// TIA Portal project "ISA_navidad" (V16)

(* hardware
DEVICE "S7-1200 station_1"  S7-1200 Station
   slot 0: "Rack_0"  S7-1200 Rack  Rack  V1.0
   slot 1: "PLC_1"  CPU 1215C DC/DC/DC  6ES7 215-1AG40-0XB0  V4.4
DEVICE "SINAMICS G_1"  Sinamics.Device
   slot 0: "	_0"  Rail  SinamicsG120RackPN
   slot 0: "Accionamiento_1"  G120 CU240E-2 PN  6SL3244-0BB12-1FA0  4.7.10
      slot 1: "Interfaz PROFINET"  MDD-SinamicsG120-P
   slot 3: "PM240 IP20"  PM240 IP20  6SL3224-0BE13-7UA0  -
DEVICE "PC-System_1"  SIMATIC PC station
   slot 0: "Estación PC SIMATIC"  Rail  SIMATIC PC-Station  V1.0
      slot 125: "Stationmanager"  Station_Manager  V6.0.4
   slot 1: "HMI_RT_1"  WinCC RT Advanced  6AV2 104-0xxxx-xxxx  16.0.0.0
      slot 33792: "Interfaz del equipo"  Host interface
   slot 2: "IE general_1"  IE General  IE_CP  V8.2.0
*)

// ===== PLC "PLC_1"  CPU 1215C DC/DC/DC =====

VAR_GLOBAL   // PLC tag table "Tabla de variables estándar"
   "marcha_pulsador" AT %I0.0 : Bool;   // S1
   "paro_pulsador" AT %I0.1 : Bool;   // S2
   "emergencia_pulsador" AT %I0.2 : Bool;   // S3
   "funcionamiento_variador" AT %I0.5 : Bool;   // DO1+ (Motor girando)
   "aviso_activo_variador" AT %I0.6 : Bool;   // DO2+ (Variador en fallo)
   "temperatura_sensor" AT %IW64 : Int;   // B4
   "nivel_sensor" AT %IW66 : Int;   // B5
   "marcha_variador" AT %Q0.0 : Bool;
   "verde_piloto" AT %Q0.1 : Bool;   // H1
   "rojo_piloto" AT %Q0.2 : Bool;   // H2
   "ambar_piloto" AT %Q0.3 : Bool;   // H3
   "electrovalvula_1" AT %Q0.6 : Bool;   // Y1
   "electrovalvula_2" AT %Q0.7 : Bool;   // Y2
   "electrovalvula_3" AT %Q1.0 : Bool;   // Y3
   "resistencia_calefactora" AT %QW64 : Int;   // R1
   "frecuencia_variador" AT %QW66 : Int;
   "etapa_0" AT %M10.0 : Bool;
   "etapa_1" AT %M10.1 : Bool;
   "etapa_2" AT %M10.2 : Bool;
   "etapa_3" AT %M10.3 : Bool;
   "etapa_4" AT %M10.4 : Bool;
   "etapa_5" AT %M10.5 : Bool;
   "etapa_10" AT %M11.0 : Bool;
   "etapa_11" AT %M11.1 : Bool;
   "etapa_12" AT %M11.2 : Bool;
   "principal_etapas" AT %MB10 : Byte;   // Etapas 0 a 5
   "System_Byte" AT %MB1 : Byte;
   "FirstScan" AT %M1.0 : Bool;
   "DiagStatusUpdate" AT %M1.1 : Bool;
   "AlwaysTRUE" AT %M1.2 : Bool;
   "AlwaysFALSE" AT %M1.3 : Bool;
   "Clock_Byte" AT %MB0 : Byte;
   "Clock_10Hz" AT %M0.0 : Bool;
   "Clock_5Hz" AT %M0.1 : Bool;
   "Clock_2.5Hz" AT %M0.2 : Bool;
   "Clock_2Hz" AT %M0.3 : Bool;
   "Clock_1.25Hz" AT %M0.4 : Bool;
   "Clock_1Hz" AT %M0.5 : Bool;
   "Clock_0.625Hz" AT %M0.6 : Bool;
   "Clock_0.5Hz" AT %M0.7 : Bool;
END_VAR

DATA_BLOCK "Variables"   // DB1
{ S7_Optimized_Access := 'TRUE' }
VERSION : 0.1
   VAR
      T1_PT : Time;   // PT de T1 convertido a segundos
      T2_PT : Time;   // PT de T2 convertido a segundos
      Setpoint_PID : Real;   // Setpoint del PID
      temperatura_escalada : Real;   // Temperatura escalada [0..100]ºC
      mode_PID : Int;   // Modo de funcionamiento PID
      mode_activate_PID : Bool;   // Activación del modo de PID
      output_PID : Real;   // Salida del PID [0..100]%
      nivel_escalado : Real;   // Nivel del tanque escalado [0..75] litros
      velocidad_lenta_SCADA : Int;   // Frecuencia lenta seleccionada en SCADA
      velocidad_rapida_SCADA : Int;   // Frecuencia rápida seleccionada en SCADA
      consigna_velocidad : Int;   // Consigna de frecuencia del variador
      paro_SCADA : Bool;   // Pulsador de paro en SCADA
      marcha_SCADA : Bool;   // Pulsador de marcha en SCADA
      estado_motor_scada : Bool;   // Piloto estado motor SCADA
      paro_emergencia_SCADA : Bool;   // Paro de emergencia SCADA
      piloto_velocidad_lenta_SCADA : Bool;   // Piloto de velocidad lenta SCADA
      piloto_velocidad_rapida_SCADA : Bool;   // Piloto de velocidad rápida SCADA
      tiempo_restante_T1 : Time;   // Tiempo restante T1
      tiempo_restante_T2 : Time;   // Tiempo restante T2
      T1_PT_ms : Time;   // PT T1 en ms introducido en SCADA
      T2_PT_ms : Time;   // PT T2 en ms introducido en SCADA
      estado_ev1 : Bool;   // Piloto estado electroválvula 1
      estado_ev2 : Bool;   // Piloto estado electroválvula 2
      estado_ev3 : Bool;   // Piloto estado electroválvula 3
      nivel_tanque1 : Time;   // Nivel del tanque A
      nivel_tanque2 : Time;   // Nivel del tanque B
      flanco_mode_activate_PID : Bool;   // Flanco de "mode_activate_PID"
      hora_activacion_SCADA : USInt;   // Hora de entrada a mantenimiento SCADA
      minuto_activacion_SCADA : USInt;   // Minuto de entrada a mantenimiento SCADA
      hora_desactivacion_SCADA : USInt;   // Hora de salida de mantenimiento SCADA
      minuto_desactivacion_SCADA_1 : USInt;   // Minuto de salida de mantenimiento SCADA
      en_mantenimiento : Bool;   // Dentro de horario de mantenimiento
      tiempo_local : DTL;   // Hora local del PLC
      estado_H1_SCADA : Bool;   // Estado piloto H1 SCADA
      estado_H2_SCADA : Bool;   // Estado piloto H2 SCADA
      estado_H3_SCADA : Bool;   // Estado piloto H3 SCADA
      simulacion_IW64 : Int;   // Simulación del sensor de temperatura
      simulacion_IW66 : Int;   // Simulación del sensor de nivel
   END_VAR
BEGIN
END_DATA_BLOCK

DATA_BLOCK "temperatura"   // DB4
{ S7_Optimized_Access := 'TRUE' }
VERSION : 0.1
// stored: InstanceOfName Analog_IN_temperatura
"Analog_IN_temperatura"
BEGIN
END_DATA_BLOCK

DATA_BLOCK "nivel"   // DB5
{ S7_Optimized_Access := 'TRUE' }
VERSION : 0.1
// stored: InstanceOfName Analog_IN_nivel
"Analog_IN_nivel"
BEGIN
END_DATA_BLOCK

DATA_BLOCK "resistencia"   // DB7
{ S7_Optimized_Access := 'TRUE' }
VERSION : 0.1
// stored: InstanceOfName Analog_OUT_resistencia
"Analog_OUT_resistencia"
BEGIN
END_DATA_BLOCK

DATA_BLOCK "frecuencia"   // DB8
{ S7_Optimized_Access := 'TRUE' }
VERSION : 0.1
// stored: InstanceOfName Analog_OUT_frecuencia
"Analog_OUT_frecuencia"
BEGIN
END_DATA_BLOCK

DATA_BLOCK "LGF_TimerSwitch_DB"   // DB9
{ S7_Optimized_Access := 'TRUE' }
AUTHOR : Siemens_Digital_Industry
FAMILY : LGF
NAME : LGF_TimerSwitch
VERSION : 0.1
// stored: InstanceOfName LGF_TimerSwitch
"LGF_TimerSwitch"
BEGIN
END_DATA_BLOCK

// folder: System blocks/Program resources

DATA_BLOCK "T1"   // DB2
{ S7_Optimized_Access := 'TRUE' }
AUTHOR : Simatic
FAMILY : IEC
NAME : IEC_TMR
VERSION : 1.0
// stored: InstanceOfName IEC_TIMER
"IEC_TIMER"
BEGIN
END_DATA_BLOCK

DATA_BLOCK "T2"   // DB3
{ S7_Optimized_Access := 'TRUE' }
AUTHOR : Simatic
FAMILY : IEC
NAME : IEC_TMR
VERSION : 1.0
// stored: InstanceOfName IEC_TIMER
"IEC_TIMER"
BEGIN
END_DATA_BLOCK

// folder: (top level)

FUNCTION_BLOCK "Analog_IN_temperatura"   // FB4, LAD
{ S7_Optimized_Access := 'TRUE' }
VERSION : 0.1
   VAR_INPUT
      Input : Int;
      X_min : Real;
      X_max : Real;
      Y_min : Real;
      Y_max : Real;
      IsTension : Bool;
   END_VAR
   VAR_OUTPUT
      Output : Real;
   END_VAR
   VAR
      X_min_bits : Int;
      X_max_bits : Int;
      norm : Real;
   END_VAR
   VAR CONSTANT
      tension_pendent : Real := 2764.8;
      intensity_pendent : Real := 1382.4;
   END_VAR
BEGIN

REGION Network 1 (SCL)

   IF #IsTension THEN
       #X_min_bits := REAL_TO_INT(#X_min * #tension_pendent);
       #X_max_bits := REAL_TO_INT(#X_max * #tension_pendent);
   ELSE
       #X_min_bits := REAL_TO_INT(#X_min * #intensity_pendent);
       #X_max_bits := REAL_TO_INT(#X_max * #intensity_pendent);
   END_IF;
END_REGION

REGION Network 2
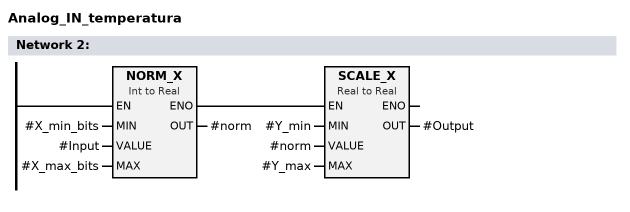
   RUNG wire#powerrail
      { S7_Templates := "[SrcType := Int, DestType := Real]" } Normalize(min := #X_min_bits, value := #Input, max := #X_max_bits, out => #norm)
      { S7_Templates := "[SrcType := Real, DestType := Real]" } Scale(min := #Y_min, value := #norm, max := #Y_max, out => #Output)
   END_RUNG
   // the same network as SCL:
   #norm := NORM_X(MIN := #X_min_bits, VALUE := #Input, MAX := #X_max_bits);
   #Output := SCALE_X(MIN := #Y_min, VALUE := #norm, MAX := #Y_max);
END_REGION
END_FUNCTION_BLOCK

FUNCTION_BLOCK "Analog_OUT_resistencia"   // FB5, LAD
{ S7_Optimized_Access := 'TRUE' }
VERSION : 0.1
   VAR_INPUT
      Input : Real;
      X_min : Real;
      X_max : Real;
      Y_min : Real;
      Y_max : Real;
      IsTension : Bool;
   END_VAR
   VAR_OUTPUT
      Output : Int;
   END_VAR
   VAR
      Y_min_bits : Int;
      Y_max_bits : Int;
      norm : Real;
   END_VAR
   VAR CONSTANT
      tension_pendent : Real := 2764.8;
      intensity_pendent : Real := 1382.4;
   END_VAR
BEGIN

REGION Network 1 (SCL)

   IF #IsTension THEN
       #Y_min_bits := REAL_TO_INT(#Y_min * #tension_pendent);
       #Y_max_bits := REAL_TO_INT(#Y_max * #tension_pendent);
   ELSE
       #Y_min_bits := REAL_TO_INT(#Y_min * #intensity_pendent);
       #Y_max_bits := REAL_TO_INT(#Y_max * #intensity_pendent);
   END_IF;
END_REGION

REGION Network 2
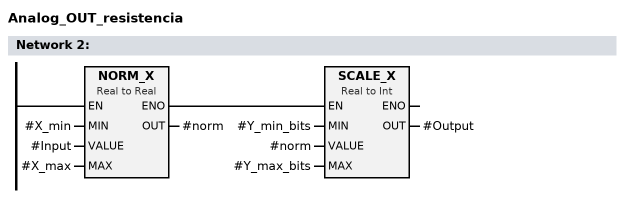
   RUNG wire#powerrail
      { S7_Templates := "[SrcType := Real, DestType := Real]" } Normalize(min := #X_min, value := #Input, max := #X_max, out => #norm)
      { S7_Templates := "[SrcType := Real, DestType := Int]" } Scale(min := #Y_min_bits, value := #norm, max := #Y_max_bits, out => #Output)
   END_RUNG
   // the same network as SCL:
   #norm := NORM_X(MIN := #X_min, VALUE := #Input, MAX := #X_max);
   #Output := SCALE_X(MIN := #Y_min_bits, VALUE := #norm, MAX := #Y_max_bits);
END_REGION
END_FUNCTION_BLOCK

FUNCTION_BLOCK "Analog_IN_nivel"   // FB6, LAD
{ S7_Optimized_Access := 'TRUE' }
VERSION : 0.1
   VAR_INPUT
      Input : Int;
      X_min : Real;
      X_max : Real;
      Y_min : Real;
      Y_max : Real;
      IsTension : Bool;
   END_VAR
   VAR_OUTPUT
      Output : Real;
   END_VAR
   VAR
      X_min_bits : Int;
      X_max_bits : Int;
      norm : Real;
   END_VAR
   VAR CONSTANT
      tension_pendent : Real := 2764.8;
      intensity_pendent : Real := 1382.4;
   END_VAR
BEGIN

REGION Network 1 (SCL)

   IF #IsTension THEN
       #X_min_bits := REAL_TO_INT(#X_min * #tension_pendent);
       #X_max_bits := REAL_TO_INT(#X_max * #tension_pendent);
   ELSE
       #X_min_bits := REAL_TO_INT(#X_min * #intensity_pendent);
       #X_max_bits := REAL_TO_INT(#X_max * #intensity_pendent);
   END_IF;
END_REGION

REGION Network 2
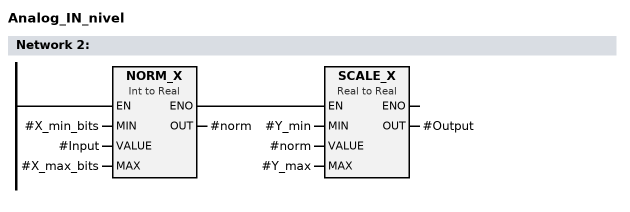
   RUNG wire#powerrail
      { S7_Templates := "[SrcType := Int, DestType := Real]" } Normalize(min := #X_min_bits, value := #Input, max := #X_max_bits, out => #norm)
      { S7_Templates := "[SrcType := Real, DestType := Real]" } Scale(min := #Y_min, value := #norm, max := #Y_max, out => #Output)
   END_RUNG
   // the same network as SCL:
   #norm := NORM_X(MIN := #X_min_bits, VALUE := #Input, MAX := #X_max_bits);
   #Output := SCALE_X(MIN := #Y_min, VALUE := #norm, MAX := #Y_max);
END_REGION
END_FUNCTION_BLOCK

FUNCTION_BLOCK "Analog_OUT_frecuencia"   // FB7, LAD
{ S7_Optimized_Access := 'TRUE' }
VERSION : 0.1
   VAR_INPUT
      Input : Real;
      X_min : Real;
      X_max : Real;
      Y_min : Real;
      Y_max : Real;
      IsTension : Bool;
   END_VAR
   VAR_OUTPUT
      Output : Int;
   END_VAR
   VAR
      Y_min_bits : Int;
      Y_max_bits : Int;
      norm : Real;
   END_VAR
   VAR CONSTANT
      tension_pendent : Real := 2764.8;
      intensity_pendent : Real := 1382.4;
   END_VAR
BEGIN

REGION Network 1 (SCL)

   IF #IsTension THEN
       #Y_min_bits := REAL_TO_INT(#Y_min * #tension_pendent);
       #Y_max_bits := REAL_TO_INT(#Y_max * #tension_pendent);
   ELSE
       #Y_min_bits := REAL_TO_INT(#Y_min * #intensity_pendent);
       #Y_max_bits := REAL_TO_INT(#Y_max * #intensity_pendent);
   END_IF;
END_REGION

REGION Network 2
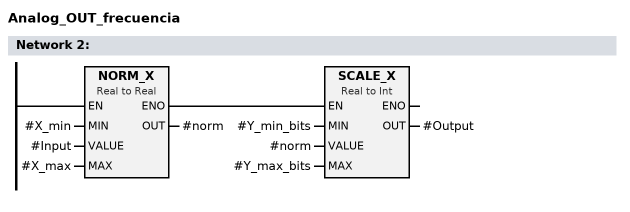
   RUNG wire#powerrail
      { S7_Templates := "[SrcType := Real, DestType := Real]" } Normalize(min := #X_min, value := #Input, max := #X_max, out => #norm)
      { S7_Templates := "[SrcType := Real, DestType := Int]" } Scale(min := #Y_min_bits, value := #norm, max := #Y_max_bits, out => #Output)
   END_RUNG
   // the same network as SCL:
   #norm := NORM_X(MIN := #X_min, VALUE := #Input, MAX := #X_max);
   #Output := SCALE_X(MIN := #Y_min_bits, VALUE := #norm, MAX := #Y_max_bits);
END_REGION
END_FUNCTION_BLOCK

ORGANIZATION_BLOCK "Principal"   // OB1, LAD, ProgramCycle
TITLE = "Main Program Sweep (Cycle)"
{ S7_Optimized_Access := 'TRUE' }
VERSION : 0.1
   VAR_INPUT
      Initial_Call : Bool;   // Initial call of this OB
      Remanence : Bool;   // =True, if remanent data are available
   END_VAR
BEGIN

REGION Network 1: Etapa 0
   // Entrar a la etapa al iniciar el sistema o cuando en la etapa 5 el tanque se vacíe por completo.
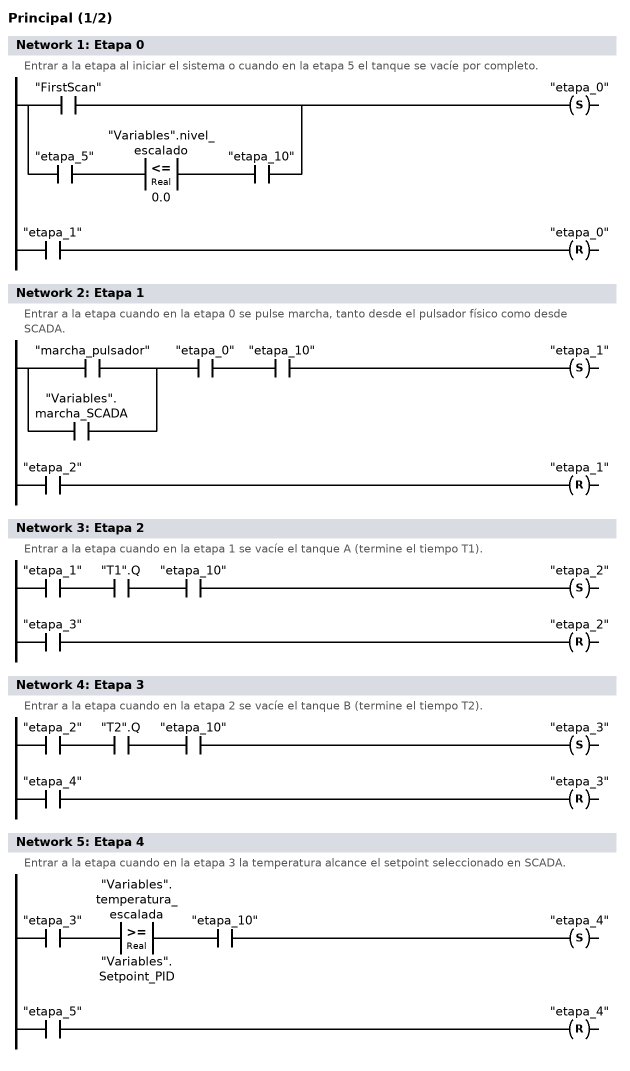
   RUNG wire#powerrail
      Contact( "FirstScan" )
      wire#w1
      S_Coil( "etapa_0" )
   END_RUNG
   RUNG wire#powerrail
      Contact( "etapa_5" )
      { S7_Templates := "SrcType := Real" } LE_Contact(in1 := "Variables".nivel_escalado, in2 := 0.0)
      Contact( "etapa_10" )
   END_RUNG wire#w1
   RUNG wire#powerrail
      Contact( "etapa_1" )
      R_Coil( "etapa_0" )
   END_RUNG
   // the same network as SCL:
   IF "FirstScan" OR ("etapa_5" AND ("Variables".nivel_escalado <= 0.0) AND "etapa_10") THEN
       "etapa_0" := TRUE;
   END_IF;
   IF "etapa_1" THEN "etapa_0" := FALSE; END_IF;
END_REGION

REGION Network 2: Etapa 1
   // Entrar a la etapa cuando en la etapa 0 se pulse marcha, tanto desde el pulsador físico como desde SCADA.
   RUNG wire#powerrail
      Contact( "marcha_pulsador" )
      wire#w1
      Contact( "etapa_0" )
      Contact( "etapa_10" )
      S_Coil( "etapa_1" )
   END_RUNG
   RUNG wire#powerrail
      Contact( "Variables".marcha_SCADA )
   END_RUNG wire#w1
   RUNG wire#powerrail
      Contact( "etapa_2" )
      R_Coil( "etapa_1" )
   END_RUNG
   // the same network as SCL:
   IF ("marcha_pulsador" OR "Variables".marcha_SCADA) AND "etapa_0" AND "etapa_10" THEN
       "etapa_1" := TRUE;
   END_IF;
   IF "etapa_2" THEN "etapa_1" := FALSE; END_IF;
END_REGION

REGION Network 3: Etapa 2
   // Entrar a la etapa cuando en la etapa 1 se vacíe el tanque A (termine el tiempo T1).
   RUNG wire#powerrail
      Contact( "etapa_1" )
      Contact( "T1".Q )
      Contact( "etapa_10" )
      S_Coil( "etapa_2" )
   END_RUNG
   RUNG wire#powerrail
      Contact( "etapa_3" )
      R_Coil( "etapa_2" )
   END_RUNG
   // the same network as SCL:
   IF "etapa_1" AND "T1".Q AND "etapa_10" THEN "etapa_2" := TRUE; END_IF;
   IF "etapa_3" THEN "etapa_2" := FALSE; END_IF;
END_REGION

REGION Network 4: Etapa 3
   // Entrar a la etapa cuando en la etapa 2 se vacíe el tanque B (termine el tiempo T2).
   RUNG wire#powerrail
      Contact( "etapa_2" )
      Contact( "T2".Q )
      Contact( "etapa_10" )
      S_Coil( "etapa_3" )
   END_RUNG
   RUNG wire#powerrail
      Contact( "etapa_4" )
      R_Coil( "etapa_3" )
   END_RUNG
   // the same network as SCL:
   IF "etapa_2" AND "T2".Q AND "etapa_10" THEN "etapa_3" := TRUE; END_IF;
   IF "etapa_4" THEN "etapa_3" := FALSE; END_IF;
END_REGION

REGION Network 5: Etapa 4
   // Entrar a la etapa cuando en la etapa 3 la temperatura alcance el setpoint seleccionado en SCADA.
   RUNG wire#powerrail
      Contact( "etapa_3" )
      { S7_Templates := "SrcType := Real" } GE_Contact(in1 := "Variables".temperatura_escalada, in2 := "Variables".Setpoint_PID)
      Contact( "etapa_10" )
      S_Coil( "etapa_4" )
   END_RUNG
   RUNG wire#powerrail
      Contact( "etapa_5" )
      R_Coil( "etapa_4" )
   END_RUNG
   // the same network as SCL:
   IF "etapa_3" AND ("Variables".temperatura_escalada >= "Variables".Setpoint_PID) AND "etapa_10" THEN
       "etapa_4" := TRUE;
   END_IF;
   IF "etapa_5" THEN "etapa_4" := FALSE; END_IF;
END_REGION

REGION Network 6: Etapa 5
   // Entrar a la etapa cuando en la etapa 4 la temperatura baje a 22ºC.
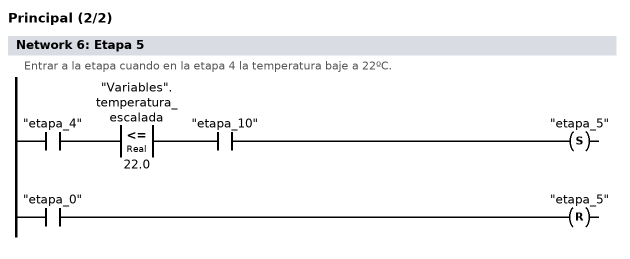
   RUNG wire#powerrail
      Contact( "etapa_4" )
      { S7_Templates := "SrcType := Real" } LE_Contact(in1 := "Variables".temperatura_escalada, in2 := 22.0)
      Contact( "etapa_10" )
      S_Coil( "etapa_5" )
   END_RUNG
   RUNG wire#powerrail
      Contact( "etapa_0" )
      R_Coil( "etapa_5" )
   END_RUNG
   // the same network as SCL:
   IF "etapa_4" AND ("Variables".temperatura_escalada <= 22.0) AND "etapa_10" THEN "etapa_5" := TRUE; END_IF;
   IF "etapa_0" THEN "etapa_5" := FALSE; END_IF;
END_REGION
END_ORGANIZATION_BLOCK

ORGANIZATION_BLOCK "PID"   // OB30, LAD, CyclicInterrupt
{ S7_Optimized_Access := 'TRUE' }
VERSION : 0.1
   VAR_INPUT
      Initial_Call : Bool;   // Initial call of this OB
      Event_Count : Int;   // Events discarded
   END_VAR
   VAR_TEMP   // added for the SCL form of the ladder/FBD networks
      _w1 : Bool;
   END_VAR
BEGIN

REGION Network 1: PID
   // Control PID que actúa sobre la resistencia calefactora para controlar la temperatura de la mezcla en el tanque.
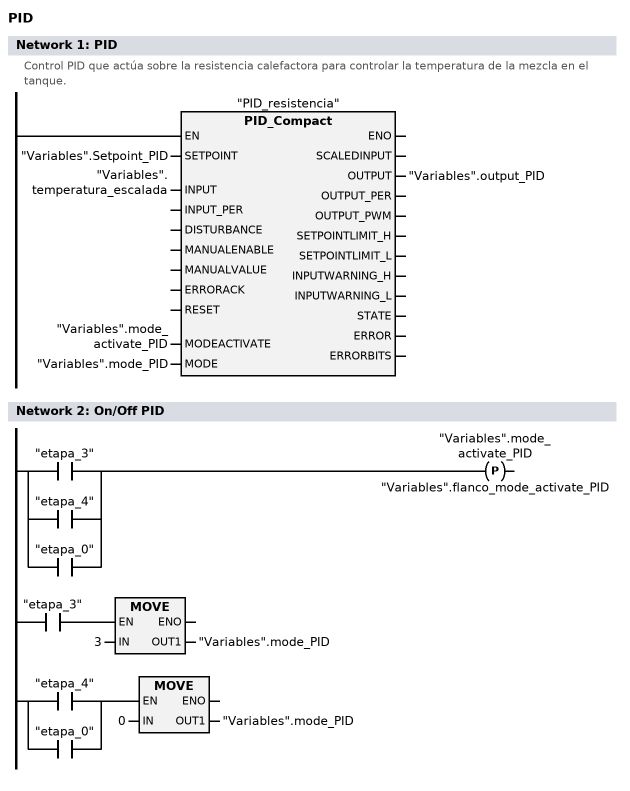
   "PID_resistencia"(Setpoint := "Variables".Setpoint_PID,   // PID_Compact
                     Input := "Variables".temperatura_escalada,
                     ModeActivate := "Variables".mode_activate_PID,
                     Mode := "Variables".mode_PID,
                     Output => "Variables".output_PID);
END_REGION

REGION Network 2: On/Off PID
   #_w1 := "etapa_3" OR "etapa_4" OR "etapa_0";
   "Variables".mode_activate_PID := #_w1 AND NOT "Variables".flanco_mode_activate_PID;   // rising edge
   "Variables".flanco_mode_activate_PID := #_w1;
   IF "etapa_3" THEN "Variables".mode_PID := 3; END_IF;
   IF "etapa_4" OR "etapa_0" THEN "Variables".mode_PID := 0; END_IF;
END_REGION

REGION Network 3 (SCL): Parámetros PID
   "PID_resistencia".Retain.CtrlParams.Gain := 10;
   "PID_resistencia".Retain.CtrlParams.Td := 10;
   "PID_resistencia".Retain.CtrlParams.Ti := 10;
END_REGION
END_ORGANIZATION_BLOCK

ORGANIZATION_BLOCK "Tratamiento Posterior"   // OB123, LAD, ProgramCycle
TITLE = "Main Program Sweep (Cycle)"
{ S7_Optimized_Access := 'TRUE' }
VERSION : 0.1
   VAR_INPUT
      Initial_Call : Bool;   // Initial call of this OB
      Remanence : Bool;   // =True, if remanent data are available
   END_VAR
BEGIN

REGION Network 1: H1
   // Indica que el motor está en funcionamiento a velocidad lenta (piloto intermitente) o rápida (piloto fijo) (para simular, "funcionamiento_variador" se considera NC pero debería ser NA).
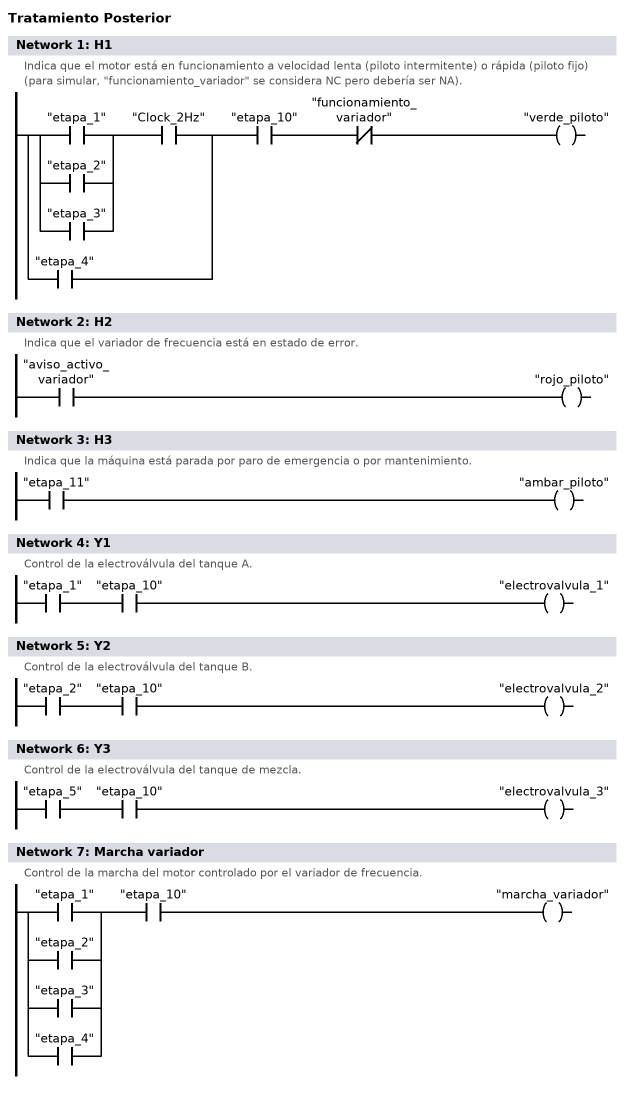
   RUNG wire#powerrail
      Contact( "etapa_1" )
      wire#w1
      Contact( "Clock_2Hz" )
      wire#w2
      Contact( "etapa_10" )
      I_Contact( "funcionamiento_variador" )
      Coil( "verde_piloto" )
   END_RUNG
   RUNG wire#powerrail
      Contact( "etapa_2" )
   END_RUNG wire#w1
   RUNG wire#powerrail
      Contact( "etapa_3" )
   END_RUNG wire#w1
   RUNG wire#powerrail
      Contact( "etapa_4" )
   END_RUNG wire#w2
   // the same network as SCL:
   "verde_piloto" := ((("etapa_1" OR "etapa_2" OR "etapa_3") AND "Clock_2Hz") OR "etapa_4") AND "etapa_10" AND NOT "funcionamiento_variador";
END_REGION

REGION Network 2: H2
   // Indica que el variador de frecuencia está en estado de error.
   RUNG wire#powerrail
      Contact( "aviso_activo_variador" )
      Coil( "rojo_piloto" )
   END_RUNG
   // the same network as SCL:
   "rojo_piloto" := "aviso_activo_variador";
END_REGION

REGION Network 3: H3
   // Indica que la máquina está parada por paro de emergencia o por mantenimiento.
   RUNG wire#powerrail
      Contact( "etapa_11" )
      Coil( "ambar_piloto" )
   END_RUNG
   // the same network as SCL:
   "ambar_piloto" := "etapa_11";
END_REGION

REGION Network 4: Y1
   // Control de la electroválvula del tanque A.
   RUNG wire#powerrail
      Contact( "etapa_1" )
      Contact( "etapa_10" )
      Coil( "electrovalvula_1" )
   END_RUNG
   // the same network as SCL:
   "electrovalvula_1" := "etapa_1" AND "etapa_10";
END_REGION

REGION Network 5: Y2
   // Control de la electroválvula del tanque B.
   RUNG wire#powerrail
      Contact( "etapa_2" )
      Contact( "etapa_10" )
      Coil( "electrovalvula_2" )
   END_RUNG
   // the same network as SCL:
   "electrovalvula_2" := "etapa_2" AND "etapa_10";
END_REGION

REGION Network 6: Y3
   // Control de la electroválvula del tanque de mezcla.
   RUNG wire#powerrail
      Contact( "etapa_5" )
      Contact( "etapa_10" )
      Coil( "electrovalvula_3" )
   END_RUNG
   // the same network as SCL:
   "electrovalvula_3" := "etapa_5" AND "etapa_10";
END_REGION

REGION Network 7: Marcha variador
   // Control de la marcha del motor controlado por el variador de frecuencia.
   RUNG wire#powerrail
      Contact( "etapa_1" )
      wire#w1
      Contact( "etapa_10" )
      Coil( "marcha_variador" )
   END_RUNG
   RUNG wire#powerrail
      Contact( "etapa_2" )
   END_RUNG wire#w1
   RUNG wire#powerrail
      Contact( "etapa_3" )
   END_RUNG wire#w1
   RUNG wire#powerrail
      Contact( "etapa_4" )
   END_RUNG wire#w1
   // the same network as SCL:
   "marcha_variador" := ("etapa_1" OR "etapa_2" OR "etapa_3" OR "etapa_4") AND "etapa_10";
END_REGION

REGION Network 8 (SCL): Variables SCADA
   // Asociaciones de las salidas físicas a pilotos que muestran su estado en el HMI (para simular, "funcionamiento_variador" se considera NC pero debería ser NA).
   "Variables".estado_motor_scada := "marcha_variador" AND NOT "funcionamiento_variador";
   "Variables".estado_ev1 := "electrovalvula_1";
   "Variables".estado_ev2 := "electrovalvula_2";
   "Variables".estado_ev3 := "electrovalvula_3";
   "Variables".estado_H1_SCADA := "verde_piloto";
   "Variables".estado_H2_SCADA := "rojo_piloto";
   "Variables".estado_H3_SCADA := "ambar_piloto";
END_REGION
END_ORGANIZATION_BLOCK

ORGANIZATION_BLOCK "Temporizadores"   // OB124, LAD, ProgramCycle
TITLE = "Main Program Sweep (Cycle)"
{ S7_Optimized_Access := 'TRUE' }
VERSION : 0.1
   VAR_INPUT
      Initial_Call : Bool;   // Initial call of this OB
      Remanence : Bool;   // =True, if remanent data are available
   END_VAR
BEGIN

REGION Network 1: T1
   // Cuenta el tiempo que tarda en vaciarse el tanque A.
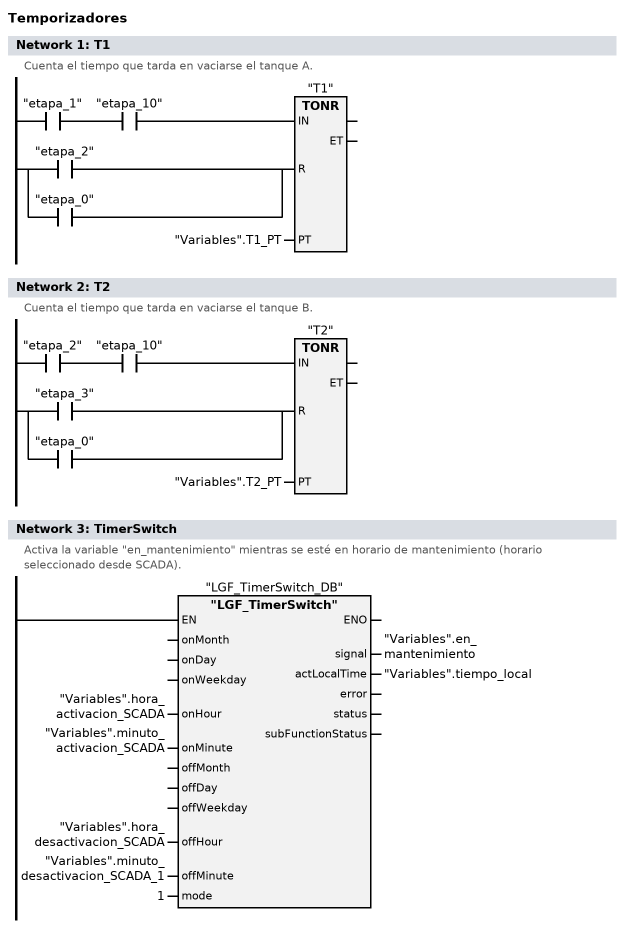
   "T1".TONR(IN := "etapa_1" AND "etapa_10", R := "etapa_2" OR "etapa_0", PT := "Variables".T1_PT);
END_REGION

REGION Network 2: T2
   // Cuenta el tiempo que tarda en vaciarse el tanque B.
   "T2".TONR(IN := "etapa_2" AND "etapa_10", R := "etapa_3" OR "etapa_0", PT := "Variables".T2_PT);
END_REGION

REGION Network 3: TimerSwitch
   // Activa la variable "en_mantenimiento" mientras se esté en horario de mantenimiento (horario seleccionado desde SCADA).
   RUNG wire#powerrail
      "LGF_TimerSwitch_DB"(onMonth :=, onDay :=, onWeekday :=, onHour := "Variables".hora_activacion_SCADA, onMinute := "Variables".minuto_activacion_SCADA, offMonth :=, offDay :=, offWeekday :=, offHour := "Variables".hora_desactivacion_SCADA, offMinute := "Variables".minuto_desactivacion_SCADA_1, mode := 1, signal => "Variables".en_mantenimiento, actLocalTime => "Variables".tiempo_local, error =>, status =>, subFunctionStatus =>)
   END_RUNG
   // the same network as SCL:
   "LGF_TimerSwitch_DB"(onHour := "Variables".hora_activacion_SCADA,   // "LGF_TimerSwitch"
                        onMinute := "Variables".minuto_activacion_SCADA,
                        offHour := "Variables".hora_desactivacion_SCADA,
                        offMinute := "Variables".minuto_desactivacion_SCADA_1,
                        mode := 1,
                        signal => "Variables".en_mantenimiento,
                        actLocalTime => "Variables".tiempo_local);
END_REGION
END_ORGANIZATION_BLOCK

ORGANIZATION_BLOCK "Escalados"   // OB125, LAD, ProgramCycle
TITLE = "Main Program Sweep (Cycle)"
{ S7_Optimized_Access := 'TRUE' }
VERSION : 0.1
// Escalados de las entradas y salidas analógicas
   VAR_INPUT
      Initial_Call : Bool;   // Initial call of this OB
      Remanence : Bool;   // =True, if remanent data are available
   END_VAR
BEGIN

REGION Network 1: Sensor de temperatura
   // Escalado de la señal [0..10]V del sensor de temperatura [0..100]ºC (para simular, la entrada IW64 es sustituida por su simulación controlada desde SCADA).
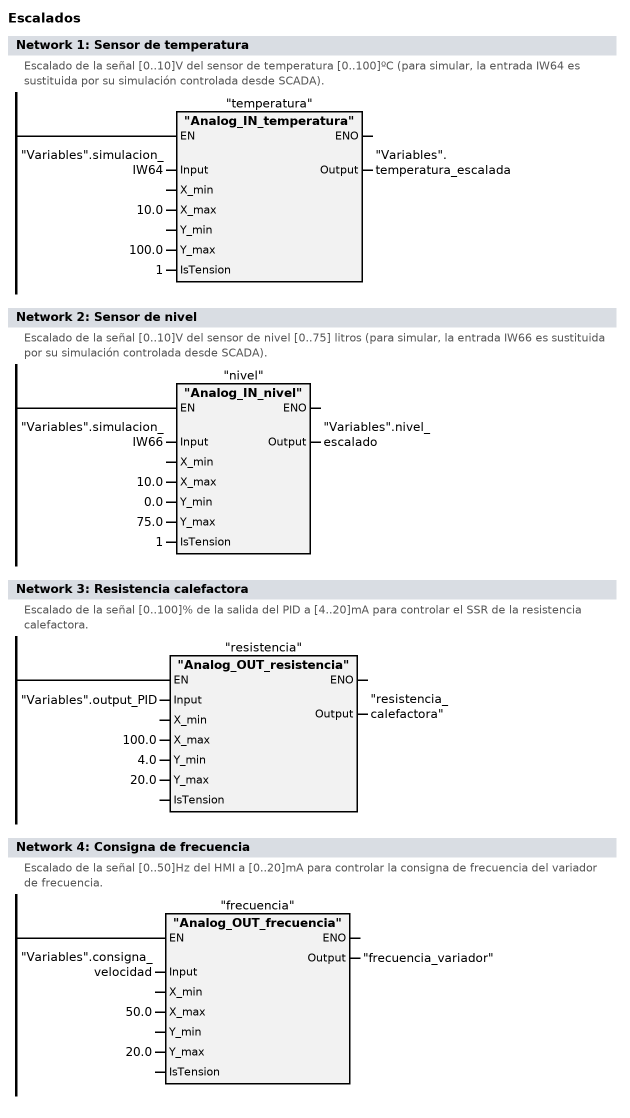
   RUNG wire#powerrail
      "temperatura"(Input := "Variables".simulacion_IW64, X_min :=, X_max := 10.0, Y_min :=, Y_max := 100.0, IsTension := 1, Output => "Variables".temperatura_escalada)
   END_RUNG
   // the same network as SCL:
   "temperatura"(Input := "Variables".simulacion_IW64,   // "Analog_IN_temperatura"
                 X_max := 10.0,
                 Y_max := 100.0,
                 IsTension := 1,
                 Output => "Variables".temperatura_escalada);
END_REGION

REGION Network 2: Sensor de nivel
   // Escalado de la señal [0..10]V del sensor de nivel [0..75] litros (para simular, la entrada IW66 es sustituida por su simulación controlada desde SCADA).
   RUNG wire#powerrail
      "nivel"(Input := "Variables".simulacion_IW66, X_min :=, X_max := 10.0, Y_min := 0.0, Y_max := 75.0, IsTension := 1, Output => "Variables".nivel_escalado)
   END_RUNG
   // the same network as SCL:
   "nivel"(Input := "Variables".simulacion_IW66,   // "Analog_IN_nivel"
           X_max := 10.0,
           Y_min := 0.0,
           Y_max := 75.0,
           IsTension := 1,
           Output => "Variables".nivel_escalado);
END_REGION

REGION Network 3: Resistencia calefactora
   // Escalado de la señal [0..100]% de la salida del PID a [4..20]mA para controlar el SSR de la resistencia calefactora.
   RUNG wire#powerrail
      "resistencia"(Input := "Variables".output_PID, X_min :=, X_max := 100.0, Y_min := 4.0, Y_max := 20.0, IsTension :=, Output => "resistencia_calefactora")
   END_RUNG
   // the same network as SCL:
   "resistencia"(Input := "Variables".output_PID,   // "Analog_OUT_resistencia"
                 X_max := 100.0,
                 Y_min := 4.0,
                 Y_max := 20.0,
                 Output => "resistencia_calefactora");
END_REGION

REGION Network 4: Consigna de frecuencia
   // Escalado de la señal [0..50]Hz del HMI a [0..20]mA para controlar la consigna de frecuencia del variador de frecuencia.
   RUNG wire#powerrail
      "frecuencia"(Input := "Variables".consigna_velocidad, X_min :=, X_max := 50.0, Y_min :=, Y_max := 20.0, IsTension :=, Output => "frecuencia_variador")
   END_RUNG
   // the same network as SCL:
   "frecuencia"(Input := "Variables".consigna_velocidad,   // "Analog_OUT_frecuencia"
                X_max := 50.0,
                Y_max := 20.0,
                Output => "frecuencia_variador");
END_REGION
END_ORGANIZATION_BLOCK

ORGANIZATION_BLOCK "Paro Emergencia / mantenimiento"   // OB126, LAD, ProgramCycle
TITLE = "Main Program Sweep (Cycle)"
{ S7_Optimized_Access := 'TRUE' }
VERSION : 0.1
// Funcionamiento paro de emergencia o por mantenimiento. Al pulsar la seta de emergencia o entrar en horario de mantenimiento, se para todo el sistema. Al rearmar la seta de emergencia y estar fuera de horario de mantenimiento, el sistema sigue desde donde se había quedado.
   VAR_INPUT
      Initial_Call : Bool;   // Initial call of this OB
      Remanence : Bool;   // =True, if remanent data are available
   END_VAR
BEGIN

REGION Network 1: Etapa 10
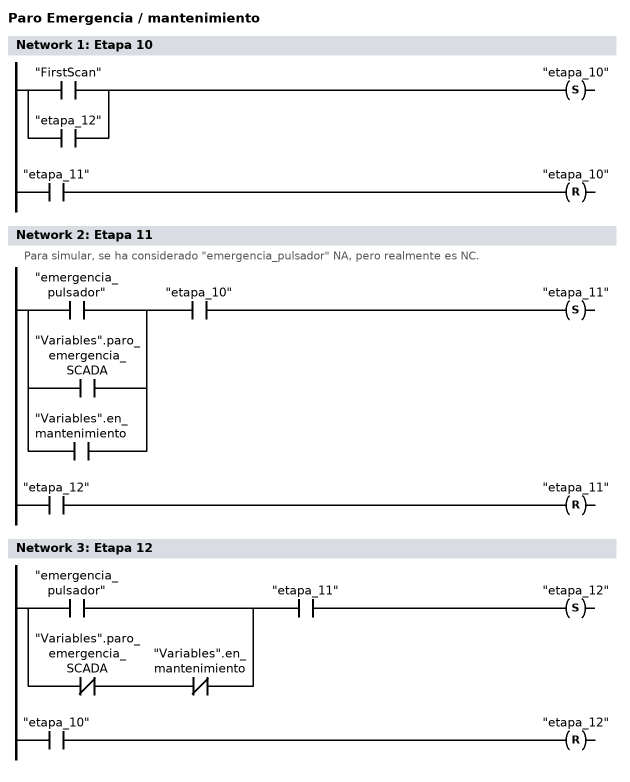
   RUNG wire#powerrail
      Contact( "FirstScan" )
      wire#w1
      S_Coil( "etapa_10" )
   END_RUNG
   RUNG wire#powerrail
      Contact( "etapa_12" )
   END_RUNG wire#w1
   RUNG wire#powerrail
      Contact( "etapa_11" )
      R_Coil( "etapa_10" )
   END_RUNG
   // the same network as SCL:
   IF "FirstScan" OR "etapa_12" THEN "etapa_10" := TRUE; END_IF;
   IF "etapa_11" THEN "etapa_10" := FALSE; END_IF;
END_REGION

REGION Network 2: Etapa 11
   // Para simular, se ha considerado "emergencia_pulsador" NA, pero realmente es NC.
   RUNG wire#powerrail
      Contact( "emergencia_pulsador" )
      wire#w1
      Contact( "etapa_10" )
      S_Coil( "etapa_11" )
   END_RUNG
   RUNG wire#powerrail
      Contact( "Variables".paro_emergencia_SCADA )
   END_RUNG wire#w1
   RUNG wire#powerrail
      Contact( "Variables".en_mantenimiento )
   END_RUNG wire#w1
   RUNG wire#powerrail
      Contact( "etapa_12" )
      R_Coil( "etapa_11" )
   END_RUNG
   // the same network as SCL:
   IF ("emergencia_pulsador" OR "Variables".paro_emergencia_SCADA OR "Variables".en_mantenimiento) AND "etapa_10" THEN
       "etapa_11" := TRUE;
   END_IF;
   IF "etapa_12" THEN "etapa_11" := FALSE; END_IF;
END_REGION

REGION Network 3: Etapa 12
   RUNG wire#powerrail
      Contact( "emergencia_pulsador" )
      wire#w1
      Contact( "etapa_11" )
      S_Coil( "etapa_12" )
   END_RUNG
   RUNG wire#powerrail
      I_Contact( "Variables".paro_emergencia_SCADA )
      I_Contact( "Variables".en_mantenimiento )
   END_RUNG wire#w1
   RUNG wire#powerrail
      Contact( "etapa_10" )
      R_Coil( "etapa_12" )
   END_RUNG
   // the same network as SCL:
   IF ("emergencia_pulsador" OR (NOT "Variables".paro_emergencia_SCADA AND NOT "Variables".en_mantenimiento)) AND "etapa_11" THEN
       "etapa_12" := TRUE;
   END_IF;
   IF "etapa_10" THEN "etapa_12" := FALSE; END_IF;
END_REGION
END_ORGANIZATION_BLOCK

ORGANIZATION_BLOCK "Paro"   // OB127, SCL, ProgramCycle
TITLE = "Main Program Sweep (Cycle)"
{ S7_Optimized_Access := 'TRUE' }
VERSION : 0.1
   VAR_INPUT
      Initial_Call : Bool;   // Initial call of this OB
      Remanence : Bool;   // =True, if remanent data are available
   END_VAR
BEGIN
   // volver a la etapa 0 si se pulsa paro (tanto desde el pulsador como desde HMI) o si se entra en horario de mantenimiento
   // (para simular, se ha considerado "paro_pulsador" NA, pero realmente es NC)
   IF "paro_pulsador" OR "Variables".paro_SCADA OR "Variables".en_mantenimiento THEN
       "principal_etapas" := 2#00000001;
   END_IF;
END_ORGANIZATION_BLOCK

ORGANIZATION_BLOCK "Calculos"   // OB130, SCL, ProgramCycle
TITLE = "Main Program Sweep (Cycle)"
{ S7_Optimized_Access := 'TRUE' }
VERSION : 0.1
   VAR_INPUT
      Initial_Call : Bool;   // Initial call of this OB
      Remanence : Bool;   // =True, if remanent data are available
   END_VAR
BEGIN
   // nivel de tanques
   "Variables".nivel_tanque1 := "T1".PT - "T1".ET;
   "Variables".nivel_tanque2 := "T2".PT - "T2".ET;

   // conversión de milisegundos a segundos
   "Variables".T1_PT := "Variables".T1_PT_ms * 1000;
   "Variables".T2_PT := "Variables".T2_PT_ms * 1000;
   "Variables".tiempo_restante_T1 := ("T1".PT - "T1".ET) / 1000;
   "Variables".tiempo_restante_T2 := ("T2".PT - "T2".ET) / 1000;

   // selección de consigna de frecuencia lenta o rápida e indicación en SCADA
   IF ("etapa_1" OR "etapa_2" OR "etapa_3") AND "marcha_variador" THEN
       "Variables".consigna_velocidad := "Variables".velocidad_lenta_SCADA;
       "Variables".piloto_velocidad_lenta_SCADA := TRUE;
       "Variables".piloto_velocidad_rapida_SCADA := FALSE;
   ELSIF "etapa_4" AND "marcha_variador" THEN
       "Variables".consigna_velocidad := "Variables".velocidad_rapida_SCADA;
       "Variables".piloto_velocidad_lenta_SCADA := FALSE;
       "Variables".piloto_velocidad_rapida_SCADA := TRUE;
   ELSE
       "Variables".consigna_velocidad := 0;
       "Variables".piloto_velocidad_lenta_SCADA := FALSE;
       "Variables".piloto_velocidad_rapida_SCADA := FALSE;
   END_IF;
END_ORGANIZATION_BLOCK

// folder: LGF/1 Date and timer operations

FUNCTION_BLOCK "LGF_TimerSwitch"   // FB10002, SCL
TITLE = LGF_TimerSwitch
{ S7_Optimized_Access := 'TRUE' }
AUTHOR : Siemens_Digital_Industry
FAMILY : LGF
NAME : LGF_TimerSwitch
// This block is a timer. It is possible to define daily, weekly, monthly, yearly time switch points and time switch points for working days or weekend days.  
// Mode: Daily: 1, weekly: 2, monthly: 3, yearly: 4, workday: 5, weekend: 6  
// 
// The time value is always compared with the local time of the PLC, therefore the time value specified at the On and Off parameters must be specified as local time.
// Dieser Baustein ist eine Zeitschaltuhr. Es ist möglich tägliche, wöchentliche, monatliche, jährliche Zeitschaltpunkte und Zeitschaltpunkte für Werktage oder Wochenendtage festzulegen.  
// Mode: Täglich: 1, Wöchentlich: 2, Monatlich: 3, Jährlich: 4, Arbeitstage: 5, Wochenende: 6  
// 
// Der Zeitwert wird immer mit der Lokalzeit der SPS verglichen, daher muss der Zeitwert, der bei den On- und Off-Parametern angegeben wird, als lokale Zeit angegeben werden.
   VAR_INPUT
      onMonth : USInt;   // Month, in which the signal shall be set. / Monat, in der der Ausgang gesetzt wird
      onDay : USInt;   // Day, at which the signal shall be set. / Tag, an dem der Ausgang gesetzt wird
      onWeekday : USInt;   // Day of the week on which the signal will be set; Sunday: 1, Monday: 2, Tuesday: 3, ... / Wochentag, an dem der Ausgang gesetzt wird; Sonntag: 1, Montag: 2, Dienstag: 3, ...
      onHour : USInt;   // Hour, at which the signal shall be set. / Stunde, in der der Ausgang gesetzt wird
      onMinute : USInt;   // Minute, at which the signal shall be set. / Minute, in der der Ausgang gesetzt wird
      offMonth : USInt;   // Month, in which the signal shall be reset. / Monat, in der der Ausgang zurückgesetzt wird
      offDay : USInt;   // Day, at which the signal shall be reset. / Tag, an dem der Ausgang zurückgesetzt wird
      offWeekday : USInt;   // Day of the week on which the signal will be reset; Sunday: 1, Monday: 2, Tuesday: 3, ... / Wochentag, an dem der Ausgang zurückgesetzt wird; Sonntag: 1, Montag: 2, Dienstag: 3, ...
      offHour : USInt;   // Hour, at which the signal shall be reset. / Stunde, in der der Ausgang zurückgesetzt wird
      offMinute : USInt;   // Minute, at which the signal shall be reset. / Minute, in der der Ausgang zurückgesetzt wird
      mode : USInt;   // Specifies the mode (see Principle of operation); Daily: 1, weekly: 2, monthly: 3, yearly: 4, workday: 5, weekend: 6 / Angabe des Modus (siehe Funktionsweise); Täglich: 1, Wöchentlich: 2, Monatlich: 3, Jährlich: 4, Arbeitstage: 5, Wochenende: 6
   END_VAR
   VAR_OUTPUT
      signal : Bool;   // Output signal / Ausagngssignal
      actLocalTime : DTL;   // Current local time / Aktuelle Lokalzeit
      error : Bool;   // FALSE: No error / TRUE: An error occurred during the execution of the FB / FALSE: Kein Fehler / TRUE: Während der Ausführung des FB ist ein Fehler aufgetreten
      status : Word;   // 16#0000-16#7FFF: Status of the FB / 16#8000-16#FFFF: Error identification (see following Table) / 16#0000-16#7FFF: Status des FB / 16#8000-16#FFFF: Fehleridentifikation (siehe folgende Tabelle)
      subFunctionStatus : Word;   // Sub function status code / Status Word einer aufgerufenen Unterfunktion
   END_VAR
   VAR_TEMP
      tempTime : DTL;   // Temp variable for current time and date read by RD_LOC_T / Temp Variable für die aktuelle Zeit und das aktuelle Datum von RD_LOC_T
      tempReadTimeStatus : Word;   // Status of the RD_LOC_T instruction / Status Wort der Systemfunktion RD_LOC_T
      tempOnTimeDtl : DTL;   // Temp variable for on time and date DTL / Temp Variable für Einschaltzeitpunkt (Zeit und Datum) DTL
      tempOnTimeTod : Time_Of_Day;   // Temp variable for on time TOD / Temp Variable für Einschaltzeitpunkt (Zeit) TOD
      tempOffTimeDtl : DTL;   // Temp variable for off time and date DTL / Temp Variable für Ausschaltzeitpunkt (Zeit und Datum) DTL
      tempOffTimeTod : Time_Of_Day;   // Temp variable for off time TOD / Temp Variable für Ausschaltzeitpunkt (Zeit) TOD
      tempActTimeDtl : DTL;   // Temp variable for current time and date DTL / Temp Variable für aktuelles Datum und aktuelle Zeit DTL
      tempActTimeTod : Time_Of_Day;   // Temp variable for current time read by RD_LOC_T / TOD / Temp Variable für aktuelles Datum und aktuelle Zeit von RD_LOC_T / TOD
   END_VAR
   VAR CONSTANT
      ZERO : USInt := 0;   // Zero contstant for initialization / Null Konstante zur Initialisierung
      CLEAR_DTL : DTL;   // Clear Date and Time with an empty tag / Lösche Datum und Zeit mit leerer Varibale
      STATUS_NO_ERROR : Word := 16#0000;   // Status: no error occurred / Status: kein Fehler aufgetreten
      ERR_NO_MODE_SELECTED : Word := 16#8200;   // Error: No suitable mode is selected, check input "mode" / Error: Kein vorhandener Mode ausgewählt, bitte Eingang `mode` prüfen
      ERR_RD_LOC_T : Word := 16#8600;   // Error in function RD_LOC_T, see in `subFunctionStatus` / Error in Funktion RD_LOC_T - weitere infos in `subFunctionStatus`
      MODE_DAILY : UInt := 1;   // Mode daily / Mode: Täglich
      MODE_WEEKLY : UInt := 2;   // Mode weekly / Mode: Wöchentlich
      MODE_MONTHLY : UInt := 3;   // Mode monthly / Mode: Monatlich
      MODE_YEARLY : UInt := 4;   // Mode yearly / Mode: Jährlich
      MODE_WEEK_DAYS : UInt := 5;   // Mode week days / Mode: Wochentage
      MODE_WEEKEND_DAYS : UInt := 6;   // Mode weekend days / Mode: Wochenend Tage
      MONTH_JANUARY : USInt := 1;   // Month January / Monat Januar
      MONTH_DECEMBER : USInt := 12;   // Month December / Monat Dezember
      DAY_MONDAY : USInt := 2;   // Day Monday / Wochentag Montag
      DAY_FRIDAY : USInt := 6;   // Day Friday / Wochentag Freitag
      DAY_SATURDAY : USInt := 7;   // Day Saturday / Wochentag Samstag
      DAY_SUNDAY : USInt := 1;   // Day Sunday / Wochentag Sonntag
      DAY_NEXT_SUNDAY : USInt := 8;   // Day Sunday / Wochentag - mächster Sonntag
      DAY_NEXT_MONDAY : USInt := 9;   // Day next Monday / Wochentag - nächster Montag
      DATE_INCREMENT : USInt := 1;   // Increment of date (month/year) / Inkremntierung für Datum (Monat oder Jahr)
      DAY_INCREMENT : Time := T#1d;   // Increment one day / Inkrementiere einen Tag
      WEEK_INCREMENT : Time := T#7d;   // Increment of 7 days = 1 week / Inkremntiere 7 Tage = 1 Woche
      DAYS_PER_WEEK : USInt := 7;   // One week = 7 days / Eine Woche = 7 Tage
      DEFAULT_YEAR : UInt := 2015;   // Default year to synchronize DTL.WEEKDAY with date / Default Jahr um im DTL Datentyp den Wochentag und das Datum zu synchronisieren
      DEFAULT_MONTH : USInt := 2;   // Default month to synchronize DTL.WEEKDAY with date / Default Monat um im DTL Datentyp den Wochentag und das Datum zu synchronisieren
   END_VAR
BEGIN
   REGION BLOCK INFO HEADER
     //===============================================================================
     // SIEMENS AG / (c)Copyright 2017
     //-------------------------------------------------------------------------------
     // Title:            LGF_TimerSwitch
     // Comment/Function: Timer Switch (daily, weekly, monthly, working days, ...)
     //                   Mode: Daily: 1, weekly: 2, monthly: 3, yearly: 4, workday: 5, weekend: 6
     // Library/Family:   LGF(Library General Functions)
     // Author:           Siemens Digital Industry Support
     // Tested with:      CPU1212C DC/DC/DC FW:V4.2
     // Engineering:      TIA Portal V14 Update 1
     // Restrictions:     ENO disabled - error handling done with error and status
     // Requirements:     PLC (S7-1200 / S7-1500)
     //-------------------------------------------------------------------------------
     // Change log table:
     // Version  | Date       | Expert in charge       | Changes applied
     //----------|------------|------------------------|------------------------------
     // 01.00.00 19.08.2015  Siemens Industry Online Support
     //                      First released version
     // 01.00.01 16.11.2015  Siemens Industry Online Support
     //                      Fix in mode 2
     // 01.01.00 23.05.2016  Siemens Industry Online Support
     //                      New mode 5 + 6
     //                      New output: actLocalTime
     // 01.01.01 02.01.2017  Siemens Industry Online Support
     //                      Upgrade: TIA V14 Update 1
     // 01.01.02 14.09.2018  Siemens Industry Online Support
     //                      Fix in modes 1, 3, 5, 6                    
     // 01.01.03 17.09.2018  Siemens Industry Online Support
     //                      Upgrade: TIA V15 Update 2
     // 01.01.04 10.10.2018  Siemens Industry Online Support
     //                      Connection to type restored
     // 01.01.05 23.11.2018  Siemens Industry Online Support
     //                      Upgrade: TIA V15.1
     // 01.01.10 13.11.2019  Simatic Systems Support
     //                      Magic numbers removed, tag naming added, code reworked
     // 03.00.00 23.04.2020  Simatic Systems Support
     //                      Set version to V3.0.0, harmonize the version of the whole library
     // 03.00.01 19.01.2020  Simatic Systems Support
     //                      Insert documentation
     //=============================================================================
   END_REGION BLOCK INFO HEADER

   REGION DESCRIPTION
     (/*NOTE
   :    The status of called commands is output in `subFunctionStatus`. In this case, the output value in `status` indicates which command caused the error. In this case, refer to the TIA Portal Online Help section for information on the respective commands.

   ---

   The block offers various timer types, which are determined in the `mode` parameter:

   * Daily timer (mode = 1)
   * Weekly timer (mode = 2)
   * Monthly timer (mode = 3)
   * Yearly timer (mode = 4)
   * Weekdays, Monday to Friday (mode = 5)
   * Weekend, Saturday and Sunday (mode = 6)

   The time value is always compared with the local time of the PLC, therefore the time value specified at the On and Off parameters must be specified as local time.

   Depending on the mode, the following formal parameters must be interconnected:

   +------+---------------------------------------+-----------------------------------------+
   | Mode | Mode                                  | Required formal parameters              |
   +======+=======================================+=========================================+
   | 1 .  | Daily timer                           | * onHour / offHour                      |
   |      |                                       | * onMinute / offMinute                  |
   +------+---------------------------------------+-----------------------------------------+
   | 2 .  | Weekly timer                          | * onWeekday / offWeekday                |
   |      |                                       | * onHour / offHour                      |
   |      |                                       | * onMinute / offMinute                  |
   +------+---------------------------------------+-----------------------------------------+
   | 3 .  | Monthly timer                         | * onDay / offDay                        |
   |      |                                       | * onHour / offHour                      |
   |      |                                       | * onMinute / offMinute                  |
   +------+---------------------------------------+-----------------------------------------+
   | 4 .  | Yearly timer                          | * onMonth / offMonth                    |
   |      |                                       | * onDay / offDay                        |
   |      |                                       | * onHour / offHour                      |
   |      |                                       | * onMinute / offMinute                  |
   +------+---------------------------------------+-----------------------------------------+
   | 5 .  | Weekdays                              | * onHour / offHour                      |
   |      |                                       | * onMinute / offMinute                  |
   +------+---------------------------------------+-----------------------------------------+
   | 6 .  | Weekend                               | * onHour / offHour                      |
   |      |                                       | * onMinute / offMinute                  |
   +------+---------------------------------------+-----------------------------------------+

   If the set start time equals the current local time of the controller, the output `signal` is set to `TRUE`. If the set switch-off time equals the current local time of the controller, the `signal` output is reset again.

   NOTE
   :    Please note that the block can be used in the “Monthly timer” modes (mode = 3) or “yearly timer” (mode = 4) the block only switches if the days that you specify at the input parameters, “onDay” and “offDay”, actually occur in this month.
   Hinweis
   :    In `subFunctionStatus` wird der Status von aufgerufenen Anweisungen ausge-geben. Der Ausgangswert in `status` gibt in diesem Fall an, welche Anweisung den Fehler verursacht hat. Holen Sie sich in diesem Fall die Informationen aus der TIA Portal Online Hilfe zu den jeweiligen Anweisungen.

   ---

   Der Baustein bietet verschiedene Arten einer Zeitschaltuhr, die im Parameter `mode` bestimmt werden

   * Tägliche Zeitschaltuhr (mode = 1)
   * Wöchentliche Zeitschaltuhr (mode = 2)
   * Monatliche Zeitschaltuhr (mode = 3)
   * Jährliche Zeitschaltuhr (mode = 4)
   * Werktags, Montag bis Freitag (mode = 5)
   * Wochenende, Samstag und Sonntag (mode = 6)

   Der Zeitwert wird immer mit der Lokalzeit der SPS verglichen, daher muss der Zeitwert, der bei den On- und Off-Parametern angegeben wird, als lokale Zeit angegeben werden.

   Abhängig vom Modus müssen folgende Formalparameter beschaltet werden:

   +------+---------------------------------------+-----------------------------------------+
   | Mode | Mode                                  | Required formal parameters              |
   +======+=======================================+=========================================+
   | 1 .  | Tägliche Zeitschaltuhr                | * onHour / offHour                      |
   |      |                                       | * onMinute / offMinute                  |
   +------+---------------------------------------+-----------------------------------------+
   | 2 .  | Wöchentlich Zeitschaltuhr             | * onWeekday / offWeekday                |
   |      |                                       | * onHour / offHour                      |
   |      |                                       | * onMinute / offMinute                  |
   +------+---------------------------------------+-----------------------------------------+
   | 3 .  | Monatliche Zeitschaltuhr              | * onDay / offDay                        |
   |      |                                       | * onHour / offHour                      |
   |      |                                       | * onMinute / offMinute                  |
   +------+---------------------------------------+-----------------------------------------+
   | 4 .  | Jährliche Zeitschaltuhr               | * onMonth / offMonth                    |
   |      |                                       | * onDay / offDay                        |
   |      |                                       | * onHour / offHour                      |
   |      |                                       | * onMinute / offMinute                  |
   +------+---------------------------------------+-----------------------------------------+
   | 5 .  | Werktags                              | * onHour / offHour                      |
   |      |                                       | * onMinute / offMinute                  |
   +------+---------------------------------------+-----------------------------------------+
   | 6 .  | Wochenende                            | * onHour / offHour                      |
   |      |                                       | * onMinute / offMinute                  |
   +------+---------------------------------------+-----------------------------------------+

   Entspricht die eingestellte Startzeit der aktuellen Lokalzeit der Steuerung, wird der Ausgang `signal` auf `TRUE` gesetzt. Entspricht die eingestellte Abschaltzeit der aktuellen Lokalzeit der Steuerung, wird der Ausgang `signal` wieder zurückgesetzt.

   Hinweis
   :    Beachten Sie, dass der Baustein in den Modi „Monatliche Zeitschaltuhr“ (mode = 3) oder „Jährliche Zeitschaltuhr“ (mode = 4) nur dann schaltet, wenn die Tage, die Sie an den Eingangsparametern „onDay“ und „offDay“ angeben, tatsächlich in diesem Monat vorkommen.*/)
   END_REGION DESCRIPTION

   REGION INITIALISATION
     // Time ON init
     #tempOnTimeDtl.HOUR := #onHour;
     #tempOnTimeDtl.MINUTE := #onMinute;
     #tempOnTimeDtl.SECOND := #ZERO;
     #tempOnTimeDtl.NANOSECOND := #ZERO;
     // Time OFF init
     #tempOffTimeDtl.HOUR := #offHour;
     #tempOffTimeDtl.MINUTE := #offMinute;
     #tempOffTimeDtl.SECOND := #ZERO;
     #tempOffTimeDtl.NANOSECOND := #ZERO;
   END_REGION

   REGION READ LOCAL TIME
     #tempReadTimeStatus := INT_TO_WORD(RD_LOC_T(#tempTime));

     // check result for error --> 16#8000 / MSB .X15
     IF #tempReadTimeStatus.%X15 THEN
       #error := TRUE;
       #status := #ERR_RD_LOC_T;
       #subFunctionStatus := #tempReadTimeStatus;
       #actLocalTime := #CLEAR_DTL;
       #signal := FALSE;
       RETURN;
     END_IF;

     // Store time of the current day
     #tempActTimeDtl := #tempTime;
     #tempActTimeTod := DTL_TO_TOD(#tempTime);
   END_REGION

   REGION TIMER SWITCH LOGIC
     CASE #mode OF
       #MODE_DAILY:
         REGION DAILY MODE
           #tempOnTimeDtl.YEAR := #tempActTimeDtl.YEAR;
           #tempOnTimeDtl.MONTH := #tempActTimeDtl.MONTH;
           #tempOnTimeDtl.WEEKDAY := #tempActTimeDtl.WEEKDAY;
           #tempOnTimeDtl.DAY := #tempActTimeDtl.DAY;
           // Store time of the on day
           #tempOnTimeTod := DTL_TO_TOD(#tempOnTimeDtl);

           #tempOffTimeDtl.YEAR := #tempActTimeDtl.YEAR;
           #tempOffTimeDtl.MONTH := #tempActTimeDtl.MONTH;
           #tempOffTimeDtl.WEEKDAY := #tempActTimeDtl.WEEKDAY;
           #tempOffTimeDtl.DAY := #tempActTimeDtl.DAY;
           // Store time of the off day
           #tempOffTimeTod := DTL_TO_TOD(#tempOffTimeDtl);

           // Timer setting - overnight
           IF #tempOnTimeTod > #tempOffTimeTod THEN
             // Increase the day of the timeOff when midnight happens
             IF #tempActTimeTod > #tempOffTimeTod THEN
               #tempOffTimeDtl := #tempOffTimeDtl + #DAY_INCREMENT;
             ELSE
               // Decrease the day of the timeOn when midnight happens
               // Activate signal from the midnight
               #tempOnTimeDtl := #tempOnTimeDtl - #DAY_INCREMENT;
             END_IF;
           END_IF;
         END_REGION

       #MODE_WEEKLY:
         REGION WEEKLY MODE             
           // Set the default date
           #tempOnTimeDtl.YEAR := #DEFAULT_YEAR;
           #tempOnTimeDtl.MONTH := #DEFAULT_MONTH;
           #tempOnTimeDtl.DAY := #onWeekday;  // Synchronize DTL.WEEKDAY with date

           #tempOnTimeTod := DTL_TO_TOD(#tempOnTimeDtl);

           #tempOffTimeDtl.YEAR := #DEFAULT_YEAR;
           #tempOffTimeDtl.MONTH := #DEFAULT_MONTH;
           #tempOffTimeDtl.DAY := #offWeekday;

           #tempOffTimeTod := DTL_TO_TOD(#tempOffTimeDtl);

           #tempActTimeDtl.YEAR := #DEFAULT_YEAR;
           #tempActTimeDtl.MONTH := #DEFAULT_MONTH;
           #tempActTimeDtl.DAY := #tempActTimeDtl.WEEKDAY;

           IF #onWeekday > #offWeekday OR
             (#onWeekday = #offWeekday AND #tempOnTimeTod > #tempOffTimeTod) THEN
             #tempOffTimeDtl.DAY := #offWeekday + #DAYS_PER_WEEK;

             IF #onWeekday > #tempActTimeDtl.WEEKDAY OR
               (#onWeekday = #offWeekday AND #tempActTimeTod < #tempOffTimeTod) THEN
               #tempActTimeDtl.DAY := #tempActTimeDtl.WEEKDAY + #DAYS_PER_WEEK;
             END_IF;
           END_IF;
         END_REGION

       #MODE_MONTHLY:
         REGION MONTHLY MODE
           #tempOnTimeDtl.YEAR := #tempActTimeDtl.YEAR;
           #tempOnTimeDtl.MONTH := #tempActTimeDtl.MONTH;
           #tempOnTimeDtl.WEEKDAY := #tempActTimeDtl.WEEKDAY;
           #tempOnTimeDtl.DAY := #onDay;

           #tempOnTimeTod := DTL_TO_TOD(#tempOnTimeDtl);

           #tempOffTimeDtl.YEAR := #tempActTimeDtl.YEAR;
           #tempOffTimeDtl.MONTH := #tempActTimeDtl.MONTH;
           #tempOffTimeDtl.WEEKDAY := #tempActTimeDtl.WEEKDAY;
           #tempOffTimeDtl.DAY := #offDay;

           #tempOffTimeTod := DTL_TO_TOD(#tempOffTimeDtl);

           // Timer setting - over new year
           IF #onDay > #offDay OR
             (#onDay = #offDay AND #tempOnTimeTod > #tempOffTimeTod) THEN
             IF #tempActTimeDtl.DAY > #offDay OR
               (#tempActTimeDtl.DAY = #offDay AND #tempActTimeTod > #tempOffTimeTod) THEN
               // Increase the month of the timeOff over new year
               IF #tempOffTimeDtl.MONTH = #MONTH_DECEMBER THEN
                 #tempOffTimeDtl.MONTH := #MONTH_JANUARY;
                 #tempOffTimeDtl.YEAR := #tempOffTimeDtl.YEAR + #DATE_INCREMENT;
               ELSE
                 #tempOffTimeDtl.MONTH := #tempOffTimeDtl.MONTH + #DATE_INCREMENT;
               END_IF;
             ELSE
               // Decrease the month of the timeOn over new year
               IF #tempOnTimeDtl.MONTH = #MONTH_JANUARY THEN
                 #tempOnTimeDtl.MONTH := #MONTH_DECEMBER;
                 #tempOnTimeDtl.YEAR := #tempOnTimeDtl.YEAR - #DATE_INCREMENT;
               ELSE
                 #tempOnTimeDtl.MONTH := #tempOnTimeDtl.MONTH - #DATE_INCREMENT;
               END_IF;

             END_IF;
           END_IF;
         END_REGION

       #MODE_YEARLY:
         REGION YEARLY MODE
           #tempOnTimeDtl.YEAR := #tempActTimeDtl.YEAR;
           #tempOnTimeDtl.MONTH := #onMonth;
           #tempOnTimeDtl.WEEKDAY := #tempActTimeDtl.WEEKDAY;
           #tempOnTimeDtl.DAY := #onDay;

           #tempOnTimeTod := DTL_TO_TOD(#tempOnTimeDtl);

           #tempOffTimeDtl.YEAR := #tempActTimeDtl.YEAR;
           #tempOffTimeDtl.MONTH := #offMonth;
           #tempOffTimeDtl.WEEKDAY := #tempActTimeDtl.WEEKDAY;
           #tempOffTimeDtl.DAY := #offDay;

           #tempOffTimeTod := DTL_TO_TOD(#tempOffTimeDtl);

           // Timer setting - over new year
           IF #onMonth > #offMonth OR
             (#onMonth = #offMonth AND #tempOnTimeTod > #tempOffTimeTod) THEN
             IF #tempActTimeDtl.MONTH > #offMonth OR
               (#tempActTimeDtl.MONTH = #offMonth AND #tempActTimeTod > #tempOffTimeTod) THEN
               // Increase the year of the timeOff when new year happens
               #tempOffTimeDtl.YEAR := #tempOffTimeDtl.YEAR + #DATE_INCREMENT;
             ELSE
               // Decrease the year of the timeOn when new year happens
               #tempOnTimeDtl.YEAR := #tempOnTimeDtl.YEAR - #DATE_INCREMENT;
             END_IF;
           END_IF;
         END_REGION

       #MODE_WEEK_DAYS:  // Working days (Monday - Friday)
         REGION WEEK DAYS MODE  
           #tempOnTimeDtl.YEAR := #DEFAULT_YEAR;
           #tempOnTimeDtl.MONTH := #DEFAULT_MONTH;
           #tempOnTimeDtl.DAY := #tempActTimeDtl.WEEKDAY;

           #tempOnTimeTod := DTL_TO_TOD(#tempOnTimeDtl);

           #tempOffTimeDtl.YEAR := #DEFAULT_YEAR;
           #tempOffTimeDtl.MONTH := #DEFAULT_MONTH;
           #tempOffTimeDtl.DAY := #tempActTimeDtl.WEEKDAY;

           #tempOffTimeTod := DTL_TO_TOD(#tempOffTimeDtl);

           #tempActTimeDtl.YEAR := #DEFAULT_YEAR;
           #tempActTimeDtl.MONTH := #DEFAULT_MONTH;
           #tempActTimeDtl.DAY := #tempActTimeDtl.WEEKDAY;

           // Timer setting - overnight
           IF #tempOnTimeTod > #tempOffTimeTod THEN
             IF #tempActTimeTod > #tempOffTimeTod THEN
               #tempOffTimeDtl := #tempOffTimeDtl + #DAY_INCREMENT;
             ELSE
               #tempOnTimeDtl := #tempOnTimeDtl - #DAY_INCREMENT;
             END_IF;
           END_IF;

           IF #tempOnTimeDtl.DAY <= #DAY_MONDAY THEN 
             #tempOnTimeDtl.DAY := #DAY_MONDAY;
           ELSIF #tempOnTimeDtl.DAY > #DAY_FRIDAY THEN 
             #tempOnTimeDtl.DAY := #DAY_FRIDAY;
           END_IF;

           IF #tempOffTimeDtl.DAY > #DAY_FRIDAY AND
             #tempOnTimeTod > #tempOffTimeTod THEN // #tempOffTime > Friday AND crossed midnight
             #tempOffTimeDtl.DAY := #DAY_SATURDAY;
           ELSIF #tempOffTimeDtl.DAY > #DAY_FRIDAY THEN
             #tempOffTimeDtl.DAY := #DAY_FRIDAY;
           END_IF;
         END_REGION

       #MODE_WEEKEND_DAYS:  // Weekend (Saturday and Sunday)    
         REGION WEEKEND DAYS MODE
           #tempOnTimeDtl.YEAR := #DEFAULT_YEAR;
           #tempOnTimeDtl.MONTH := #DEFAULT_MONTH;
           #tempOnTimeDtl.DAY := #tempActTimeDtl.WEEKDAY;

           IF #tempOnTimeDtl.DAY < #DAY_SATURDAY THEN
             #tempOnTimeDtl := #tempOnTimeDtl + #WEEK_INCREMENT;
           END_IF;

           #tempOnTimeTod := DTL_TO_TOD(#tempOnTimeDtl);

           #tempOffTimeDtl.YEAR := #DEFAULT_YEAR;
           #tempOffTimeDtl.MONTH := #DEFAULT_MONTH;
           #tempOffTimeDtl.DAY := #tempActTimeDtl.WEEKDAY;

           IF #tempOffTimeDtl.DAY < #DAY_SATURDAY THEN
             #tempOffTimeDtl := #tempOffTimeDtl + #WEEK_INCREMENT;
           END_IF;

           #tempOffTimeTod := DTL_TO_TOD(#tempOffTimeDtl);

           #tempActTimeDtl.YEAR := #DEFAULT_YEAR;
           #tempActTimeDtl.MONTH := #DEFAULT_MONTH;
           #tempActTimeDtl.DAY := #tempActTimeDtl.WEEKDAY;

           IF #tempActTimeDtl.DAY < #DAY_SATURDAY THEN
             #tempActTimeDtl := #tempActTimeDtl + #WEEK_INCREMENT;
           END_IF;

           #tempActTimeTod := DTL_TO_TOD(#tempTime);

           // Timer setting - overnight
           IF #tempOnTimeTod > #tempOffTimeTod THEN
             IF #tempActTimeTod > #tempOffTimeTod THEN
               #tempOffTimeDtl := #tempOffTimeDtl + #DAY_INCREMENT;
             ELSE
               #tempOnTimeDtl := #tempOnTimeDtl - #DAY_INCREMENT;
             END_IF;
           END_IF;

           IF #tempOnTimeDtl.DAY < #DAY_SATURDAY THEN
             #tempOnTimeDtl.DAY := #DAY_SATURDAY;
           ELSIF #tempOnTimeDtl.DAY > #DAY_NEXT_SUNDAY THEN
             #tempOnTimeDtl.DAY := #DAY_NEXT_SUNDAY;
           END_IF;

           IF #tempOffTimeDtl.DAY > #DAY_NEXT_SUNDAY AND
             #tempOnTimeTod > #tempOffTimeTod THEN // #tempOffTime.DAY > Sunday AND crossed midnight
             #tempOffTimeDtl.DAY := #DAY_NEXT_MONDAY;
           ELSIF #tempOffTimeDtl.DAY > #DAY_NEXT_SUNDAY THEN
             #tempOffTimeDtl.DAY := #DAY_NEXT_SUNDAY;
           END_IF;
         END_REGION
       ELSE
         #signal := FALSE;
         #actLocalTime := #CLEAR_DTL;
         #error := TRUE;
         #status := #ERR_NO_MODE_SELECTED;
         #subFunctionStatus := USINT_TO_WORD(#mode);
         RETURN;
     END_CASE;

   END_REGION

   REGION OUTPUT
     #actLocalTime := #tempTime;
     #signal := (#tempActTimeDtl >= #tempOnTimeDtl) AND (#tempActTimeDtl < #tempOffTimeDtl);
     #error := false;
     #status := #STATUS_NO_ERROR;
     #subFunctionStatus := #STATUS_NO_ERROR;

     // ENO is not used, forced to TRUE
     ENO := TRUE;
   END_REGION
END_FUNCTION_BLOCK

(* ===== HMI "HMI_RT_1" =====
system functions are stored by id; their names below are inferred from use
connection "HMI_Conexión_1": ETHERNET, S7_1200_OMS

HMI tags "Tabla de variables estándar"
   "SCADA_T1_PT" : Time = PLC Variables.T1_PT, 1 s
   "SCADA_T2_PT" : Time = PLC Variables.T2_PT, 1 s
   "Variables_consigna_velocidad" : Int = PLC Variables.consigna_velocidad, 1 s
   "Variables_velocidad_lenta_SCADA" : Int = PLC Variables.velocidad_lenta_SCADA, 1 s
   "Variables_velocidad_rapida_SCADA" : Int = PLC Variables.velocidad_rapida_SCADA, 1 s
   "Variables_paro_SCADA" : Bool = PLC Variables.paro_SCADA, 1 s
   "Variables_marcha_SCADA" : Bool = PLC Variables.marcha_SCADA, 1 s
   "Variables_paro_emergencia_SCADA" : Bool = PLC Variables.paro_emergencia_SCADA, 1 s
   "Variables_estado_motor_scada" : Bool = PLC Variables.estado_motor_scada, 1 s
   "Variables_piloto_velocidad_lenta_SCADA" : Bool = PLC Variables.piloto_velocidad_lenta_SCADA, 1 s
   "Variables_piloto_velocidad_rapida_SCADA" : Bool = PLC Variables.piloto_velocidad_rapida_SCADA, 1 s
   "Variables_tiempo_restante_T2" : Time = PLC Variables.tiempo_restante_T2, 1 s
   "T2_PT" : Time = PLC T2.PT, 1 s
   "T1_PT" : Time = PLC T1.PT, 1 s
   "Variables_tiempo_restante_T1" : Time = PLC Variables.tiempo_restante_T1, 1 s
   "Variables_T1_PT_ms" : Time = PLC Variables.T1_PT_ms, 1 s
   "Variables_T2_PT_ms" : Time = PLC Variables.T2_PT_ms, 1 s
   "Variables_estado_ev1" : Bool = PLC Variables.estado_ev1, 1 s
   "Variables_estado_ev2" : Bool = PLC Variables.estado_ev2, 1 s
   "Variables_estado_ev3" : Bool = PLC Variables.estado_ev3, 1 s
   "Variables_nivel_escalado" : Real = PLC Variables.nivel_escalado, 1 s
   "Variables_temperatura_escalada" : Real = PLC Variables.temperatura_escalada, 1 s
   "Variables_Setpoint_PID" : Real = PLC Variables.Setpoint_PID, 1 s
   "Variables_output_PID" : Real = PLC Variables.output_PID, 1 s
   "Variables_nivel_tanque1" : Time = PLC Variables.nivel_tanque1, 1 s
   "Variables_nivel_tanque2" : Time = PLC Variables.nivel_tanque2, 1 s
   "Variables_tiempo_local_HOUR" : USInt = PLC Variables.tiempo_local.HOUR, 1 s
   "Variables_tiempo_local_MINUTE" : USInt = PLC Variables.tiempo_local.MINUTE, 1 s
   "Variables_hora_activacion_SCADA" : USInt = PLC Variables.hora_activacion_SCADA, 1 s
   "Variables_hora_desactivacion_SCADA" : USInt = PLC Variables.hora_desactivacion_SCADA, 1 s
   "Variables_minuto_activación_SCADA" : USInt = PLC Variables.minuto_activacion_SCADA, 1 s
   "Variables_minuto_desactivacion_SCADA_1" : USInt = PLC Variables.minuto_desactivacion_SCADA_1, 1 s
   "Variables_estado_H1_SCADA" : Bool = PLC Variables.estado_H1_SCADA, 1 s
   "Variables_estado_H2_SCADA" : Bool = PLC Variables.estado_H2_SCADA, 1 s
   "Variables_estado_H3_SCADA" : Bool = PLC Variables.estado_H3_SCADA, 1 s
   "Variables_simulacion_IW64" : Int = PLC Variables.simulacion_IW64, 1 s
   "Variables_simulacion_IW66" : Int = PLC Variables.simulacion_IW66, 1 s

screen "Main" 1280x800
   GraphicView "Visor de gráficos_11" at 267,405 size 268x260; Picture "Gráfico_23"
   Bar "Barra_3" at 286,453 size 230x170; MinimumValue 0; MaximumValue 75
      ProcessValue <- "Variables_nivel_escalado"
   TextField "Campo de texto_1" at 846,315 size 398x26; Text 'Valor de preselección de temporizadores PT'
   TextField "Campo de texto_2" at 903,364 size 157x26; Text 'Temporizador Y1'
   IOField "Campo ES_1" at 1089,362 size 61x30; FormatPattern 99; Unit     S
      ProcessValue <- "Variables_T1_PT_ms"
   TextField "Campo de texto_3" at 903,414 size 157x26; Text 'Temporizador Y2'
   IOField "Campo ES_2" at 1089,412 size 61x30; FormatPattern 99; Unit     S
      ProcessValue <- "Variables_T2_PT_ms"
   TextField "Campo de texto_4" at 1099,41 size 105x26; Text 'Frecuencia'
   Gauge "Indicador gauge_1" at 1063,78 size 185x185; CaptionText 'SIMATIC'; UnitText 'Unit'
      ProcessValue <- "Variables_consigna_velocidad"
   TextField "Campo de texto_5" at 868,465 size 353x26; Text 'Valor de velocidad lenta y rápida en Hz'
   GraphicView "Visor de gráficos_7" at 124,14 size 139x261; Picture "Gráfico_18"
   Slider "Deslizador_1" at 932,508 size 80x261; Caption 'SIMATIC'
      ProcessValue <- "Variables_velocidad_lenta_SCADA"
   Slider "Deslizador_2" at 1077,508 size 80x261; Caption 'SIMATIC'
      ProcessValue <- "Variables_velocidad_rapida_SCADA"
   Bar "Barra_1" at 143,60 size 100x113; MinimumValue 0; MaximumValue 100
      MaximumValue <- "T1_PT"
      ProcessValue <- "Variables_nivel_tanque1"
   GraphicView "Visor de gráficos_8" at 539,13 size 139x261; Picture "Gráfico_18"
   Bar "Barra_2" at 559,59 size 100x113; MinimumValue 0; MaximumValue 100
      MaximumValue <- "T2_PT"
      ProcessValue <- "Variables_nivel_tanque2"
   Button "Botón_1" at 271,138 size 118x32; TextOff 'Paro HMI'
      on Press: SetBit("Variables_paro_SCADA")
      on Release: ResetBit("Variables_paro_SCADA")
   Button "Botón_2" at 411,138 size 118x32; TextOff 'Marcha HMI'
      on Press: SetBit("Variables_marcha_SCADA")
      on Release: ResetBit("Variables_marcha_SCADA")
   Switch "Pushbutton_Emergency" at 367,182 size 63x63; CaptionText 'Switch'; TextOff '0'; TextOn '1'; PictureOff "Pushbutton_Emergency_Off_256c"; PictureOn "Pushbutton_Emergency_On_256c"
      on Change: InvertBit("Variables_paro_emergencia_SCADA")
   Rectangle "Rectángulo_1" at 351,250 size 92x24
      Appearance <- "Variables_estado_motor_scada"
   TextField "Campo de texto_6" at 368,249 size 58x26; Text 'Motor'
      Appearance <- "Variables_estado_motor_scada"
   Rectangle "Rectángulo_2" at 268,249 size 84x25
      Appearance <- "Variables_piloto_velocidad_lenta_SCADA"
   TextField "Campo de texto_7" at 287,251 size 47x22; Text 'Lenta'
      Appearance <- "Variables_estado_motor_scada"
   Rectangle "Rectángulo_3" at 443,249 size 88x25
      Appearance <- "Variables_piloto_velocidad_rapida_SCADA"
   TextField "Campo de texto_8" at 459,251 size 57x22; Text 'Rápida'
      Appearance <- "Variables_estado_motor_scada"
   GraphicView "Visor de gráficos_12" at 175,281 size 32x68; Picture "Gráfico_24"
   GraphicView "Visor de gráficos_9" at 172,265 size 40x21; Picture "Gráfico_22"
   GraphicView "Visor de gráficos_14" at 594,281 size 32x63; Picture "Gráfico_24"
   GraphicView "Visor de gráficos_10" at 590,265 size 40x21; Picture "Gráfico_22"
   GraphicView "Visor de gráficos_1" at 181,339 size 38x38; Picture "Gráfico_28"
   GraphicView "Visor de gráficos_15" at 585,338 size 35x39; Picture "Gráfico_29"
   GraphicView "Visor de gráficos_18" at 225,350 size 49x34; Picture "Gráfico_31"
   GraphicView "Visor de gráficos_17" at 212,355 size 16x24; Picture "Gráfico_30"
   GraphicView "Visor de gráficos_20" at 528,350 size 49x34; Picture "Gráfico_31"
   GraphicView "Visor de gráficos_22" at 574,355 size 15x24; Picture "Gráfico_32"
   GraphicView "Visor de gráficos_23" at 282,357 size 36x36; Picture "Gráfico_33"
   GraphicView "Visor de gráficos_19" at 271,355 size 15x24; Picture "Gráfico_32"
   GraphicView "Visor de gráficos_24" at 292,389 size 32x38; Picture "Gráfico_24"
   GraphicView "Visor de gráficos_25" at 297,423 size 23x17; Picture "Gráfico_34"
   GraphicView "Visor de gráficos_16" at 596,293 size 57x53; Picture "qkg05uee.120"
   GraphicView "Visor de gráficos_13" at 149,294 size 58x53; Picture "xsd2twr5.rud"
   GraphicView "Visor de gráficos_26" at 484,357 size 36x40; Picture "Gráfico_35"
   GraphicView "Visor de gráficos_21" at 515,355 size 16x24; Picture "Gráfico_30"
   GraphicView "Visor de gráficos_27" at 477,390 size 32x37; Picture "Gráfico_24"
   GraphicView "Visor de gráficos_28" at 482,424 size 23x17; Picture "Gráfico_34"
   GraphicView "Visor de gráficos_29" at 355,286 size 88x127; Picture "0di04x30.usj"
   GraphicView "Visor de gráficos_4" at 343,404 size 109x175; Picture "Gráfico_13"
   GraphicView "Visor de gráficos_3" at 282,461 size 61x54; Picture "Gráfico_38"
   GraphicView "Visor de gráficos_30" at 459,573 size 59x52; Picture "n4do02ga.hq0"
   GraphicView "Visor de gráficos_5" at 450,450 size 112x36; Picture "5fvudpry.pbe"
   GraphicView "Visor de gráficos_2" at 238,592 size 95x34; Picture "awovuyyv.ole"
   GraphicView "Visor de gráficos_31" at 382,667 size 32x87; Picture "Gráfico_24"
   GraphicView "Visor de gráficos_32" at 356,680 size 58x53; Picture "xsd2twr5.rud"
   TextField "Campo de texto_9" at 363,764 size 67x26; Text 'Mezcla'
      Appearance <- "Variables_estado_motor_scada"
   GraphicView "Visor de gráficos_33" at 386,750 size 23x17; Picture "Gráfico_34"
   GraphicView "Visor de gráficos_6" at 378,652 size 40x21; Picture "Gráfico_22"
   IOField "Campo ES_3" at 712,304 size 61x30; FormatPattern 99; Unit     S
      ProcessValue <- "Variables_tiempo_restante_T2"
   IOField "Campo ES_4" at 23,304 size 61x30; FormatPattern 99; Unit     S
      ProcessValue <- "Variables_tiempo_restante_T1"
   Rectangle "Rectángulo_5" at 101,309 size 35x24
      Appearance <- "Variables_estado_ev1"
   TextField "Campo de texto_10" at 105,308 size 28x26; Text 'Y1'
      Appearance <- "Variables_estado_motor_scada"
   Rectangle "Rectángulo_6" at 664,309 size 35x24
      Appearance <- "Variables_estado_ev2"
   TextField "Campo de texto_11" at 668,308 size 28x26; Text 'Y2'
      Appearance <- "Variables_estado_motor_scada"
   Rectangle "Rectángulo_7" at 314,694 size 35x24
      Appearance <- "Variables_estado_ev3"
   TextField "Campo de texto_12" at 318,693 size 28x26; Text 'Y3'
      Appearance <- "Variables_estado_motor_scada"
   IOField "Campo ES_5" at 118,592 size 111x30; FormatPattern 99.9; Unit     litros
      ProcessValue <- "Variables_nivel_escalado"
   IOField "Campo ES_6" at 570,454 size 99x30; FormatPattern 999.9; Unit     ºC
      ProcessValue <- "Variables_temperatura_escalada"
   TextField "Campo de texto_13" at 622,493 size 211x26; Text 'Temperatura Simulada'
   TextField "Campo de texto_14" at 658,643 size 138x26; Text 'Nivel Simulado'
   TextField "Campo de texto_15" at 742,41 size 262x26; Text 'Consigna de temperatura SP'
   IOField "Campo ES_7" at 824,78 size 99x30; FormatPattern 999.9; Unit     ºC
      ProcessValue <- "Variables_Setpoint_PID"
   IOField "Campo ES_8" at 163,465 size 99x30; FormatPattern 999.9; Unit     %
      ProcessValue <- "Variables_output_PID"
   Slider "Deslizador_3" at 582,525 size 282x70; Caption 'SIMATIC'
      ProcessValue <- "Variables_simulacion_IW64"
   Slider "Deslizador_4" at 582,675 size 282x69; Caption 'SIMATIC'
      ProcessValue <- "Variables_simulacion_IW66"
   TextField "Campo de texto_16" at 750,134 size 243x26; Text 'Horario de mantenimiento'
   IOField "Campo ES_9" at 859,171 size 60x30; FormatPattern 99; Unit     h
      ProcessValue <- "Variables_hora_activacion_SCADA"
   TextField "Campo de texto_17" at 751,173 size 98x26; Text 'Activación'
   TextField "Campo de texto_18" at 719,215 size 131x26; Text 'Desactivación'
   IOField "Campo ES_11" at 925,171 size 78x30; FormatPattern 99; Unit     min
      ProcessValue <- "Variables_minuto_activación_SCADA"
   IOField "Campo ES_10" at 859,213 size 60x30; FormatPattern 99; Unit     h
      ProcessValue <- "Variables_hora_desactivacion_SCADA"
   IOField "Campo ES_12" at 925,213 size 78x30; FormatPattern 99; Unit     min
      ProcessValue <- "Variables_minuto_desactivacion_SCADA_1"
   TextField "Campo de texto_19" at 353,23 size 96x26; Text 'Hora local'
   IOField "Campo ES_13" at 330,59 size 60x30; FormatPattern 99; Unit     h
      ProcessValue <- "Variables_tiempo_local_HOUR"
   IOField "Campo ES_14" at 396,59 size 78x30; FormatPattern 99; Unit     min
      ProcessValue <- "Variables_tiempo_local_MINUTE"
   Circle "Círculo_1" at 37,30 size 48x48
      Appearance <- "Variables_estado_H1_SCADA"
   TextField "Campo de texto_20" at 46,41 size 30x26; Text 'H1'
      Appearance <- "Variables_estado_motor_scada"
   Circle "Círculo_2" at 37,97 size 48x48
      Appearance <- "Variables_estado_H2_SCADA"
   TextField "Campo de texto_21" at 46,108 size 30x26; Text 'H2'
      Appearance <- "Variables_estado_motor_scada"
   Circle "Círculo_3" at 37,164 size 48x48
      Appearance <- "Variables_estado_H3_SCADA"
   TextField "Campo de texto_22" at 46,175 size 30x26; Text 'H3'
      Appearance <- "Variables_estado_motor_scada"
*)